(* Schneider Machine Expert - Basic project simple drum to turn on 4 pumps upgraded, file version 2.7.0.0 *)
(* ProjectInformations: Name=New project *)

HARDWARE
  Cpu 0: TM221M16R/G
  EthernetConfiguration: NetworkName=M221, IpAllocationMode=FixedAddress, IpAddress=0.0.0.0, SubnetMask=0.0.0.0
  SerialLineConfiguration: Baud=Baud19200, Parity=ParityEven, DataBits=DataBits8, StopBits=StopBits1, PhysicalMedium=PhysicalMediumRs485, TransmissionMode=TransmissionModeModbusRtu, SlaveId=1, Addressing=SlaveAddressing
  MastTask: UsePeriodScanMode=false, PeriodScan=100
  FastTask: Period=255
  CpuBehavior: StartingMode=StartAsPreviousState, AutoSaveRamOnEeprom=true, WatchdogPeriod=250

SYMBOLS  (address, symbol, comment, settings)
  %M0       FULL
  %DR0        "DRUM TO PUMPS"  [Bits(BitForDrum(Outputs=%Q0.0), BitForDrum(Outputs=%Q0.1), BitForDrum(Outputs=%Q0.2), BitForDrum(Outputs=%Q0.3)), StepsNumber=5]
  %I0.0     MODE
  %I0.1     RESET

POU New POU
  (* SectionNumber=1 *)

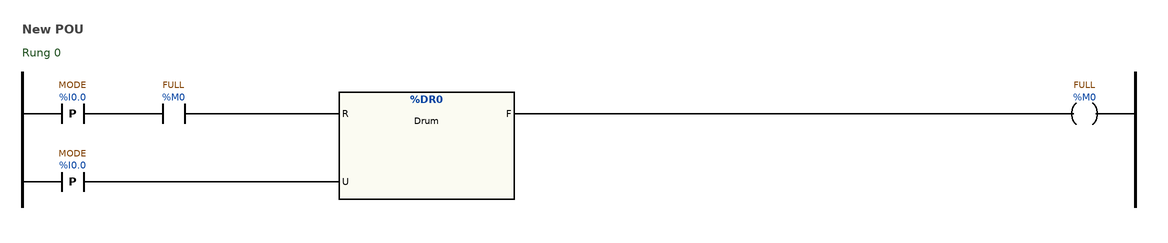

// Rung 0
  BLK %DR0
  LDR %I0.0               (* MODE *)
  AND %M0                 (* FULL *)
  R
  LDR %I0.0               (* MODE *)
  U
  OUT_BLK
  LD F
  ST %M0                  (* FULL *)
  END_BLK
  // as ST:
  //   %DR0(R := RISING(MODE) AND FULL, U := RISING(MODE));
  //   FULL := %DR0.F;
